PROGRAM ManualRotAxis
VAR
END_VAR

RAVL.axis.ReadStatus();

IF RAVL.clockwise AND NOT(RAVL.endStop) THEN
	RAVL.lastClockwise := TRUE;
	RAVL.lastCounterClockwise := FALSE;
END_IF

IF RAVL.counterClockwise AND NOT(RAVL.endStop) THEN
	RAVL.lastClockwise := FALSE;
	RAVL.lastCounterClockwise := TRUE;
END_IF

RAVL.axisPower(
	Axis:= RAVL.axis,
	Enable:= RAVL.enable,
	Enable_Positive:= RAVL.enable,
	Enable_Negative:= RAVL.enable,
	Override:= RAVL.override,
	BufferMode:= ,
	Options:= ,
	Status=> RAVL.running,
	Busy=> ,
	Active=> ,
	Error=> ,
	ErrorID=> RAVL.currentError
);

RAVL.axisMoveManual(
	Axis:= RAVL.axis,
	JogForward:= (RAVL.counterClockwise AND (NOT(RAVL.endStop) OR (RAVL.endStop AND RAVL.lastClockwise))),
	JogBackwards:= (RAVL.clockwise AND (NOT(RAVL.endStop) OR (RAVL.endStop AND RAVL.lastCounterClockwise))),
	Mode:= ,
	Position:= ,
	Velocity:= ,
	Acceleration:= ,
	Deceleration:= ,
	Jerk:= ,
	Done=> RAVL.done,
	Busy=> RAVL.busy,
	Active=> ,
	CommandAborted=> ,
	Error=> ,
	ErrorID=> RAVL.currentError
);

IF RAVL.busy THEN
	RAVL.axisReadActualPosition(Axis := RAVL.axis, Enable := TRUE, Valid=>, Busy=>, Error=>, ErrorID=>, Position=> RAVL.actualPosition);
END_IF
RAVL.actualPositionInt := LREAL_TO_INT(RAVL.actualPosition);

RAVL.axisErrorReset(Axis := RAVL.axis, Execute := RAVL.resetError, Done =>, Error =>, ErrorID => RAVL.currentError);

END_PROGRAM

(* stored: Version 1.1.0.1, ProductVersion 3.1.4024.6
   POU ManualRotAxis: Id {e5fa7945-e802-46a9-800f-6db9cf40bcd4}, SpecialFunc None *)
